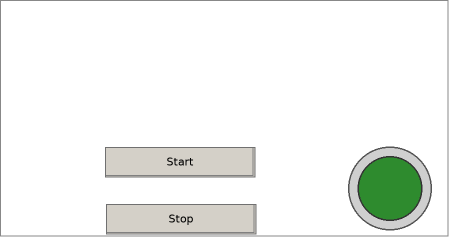
VISUALIZATION Visualization  // 449x237
    Button (105,147 150x30), "Start"
        OnMouseDown: execute { MAIN.bStartMotor := TRUE; }
        OnMouseUp: execute { MAIN.bStartMotor :=  FALSE; }
    Button (106,204 150x30), "Stop", pressed state: MAIN.bStopMotor
        OnMouseDown: execute { MAIN.bStopMotor := TRUE; }
        OnMouseUp: execute { MAIN.bStopMotor := FALSE; }
    Lamp1 (331,140 118x97), variable: MAIN.bServoMotor, style: Lamp-Lamp1-Green
END_VISUALIZATION

(* stored: Version 1.1.0.1, ProductVersion 3.1.4024.13
   Visu Visualization: Id {d761737a-16fe-4bb3-be17-d8e10b44a1d3} *)
